Staubli VAL3: setXaxis.pgx

program setXaxis()
begin
  numMessage[4]=0
  stringXarray=""
  while numMessage[4]==0
    sioGet(sioASCII,numMessage)
    stringXarray=chr(numMessage[0])
    if chr(numMessage[1])!="#"
      stringXarray=stringXarray+chr(numMessage[1])
    endIf
    toNum(stringXarray,numXarray,isNum)
    putln(stringXarray)
  endWhile
end
